TYPE ST_MachineConfig  :
STRUCT
	iDrumSpeed : INT;
	iWaterTemperature : INT;
END_STRUCT
END_TYPE

(* stored: Version 1.1.0.1, ProductVersion 3.1.4024.16
   DUT ST_MachineConfig: Id {f61cd767-f422-4c4b-a643-35e9247afc5d} *)
